# B&R Automation Studio project br_server
Automation Studio 4.4.6.71 SP

## Configuration minimal

### Task classes (Cpu.sw)
```
Cyclic#4:
  TCP_Server <- TcpIpServer.prg
Cyclic#7:
  ControlLoo <- ControlLoop.prg
Libraries: AsBrStr, AsIOTime, AsTCP, runtime, TcpIp, Transport
```

### Hardware
```
X20CP1586 : X20CP1586 v1.4.2.0
  Connector IF2:
    ActivateDevice = 1
    Mode = Manual
    InternetAddress = 10.4.22.176
    SubnetMask = 255.255.255.0
  ConfigurationID = br_server_minimal
  SimulationIPAddress = 10.4.22.176
```

## Logical view

Binary libraries used (declarations not repeated): operator, runtime, astime, AsIecCon, AsBrStr, AsIOTime, AsTCP

### Global.typ - Global data types
```iecst
TYPE
	_expData : 	STRUCT
		bActivateExperiment : BOOL;
	END_STRUCT;
	_trajData : 	STRUCT
		dStartValue : LREAL;
		lStartTime : UDINT;
		dEndValue : LREAL;
		lEndTime : UDINT;
		dOutput : LREAL;
	END_STRUCT;
	_benchData : 	STRUCT
		lTime : UDINT;
		dValue1 : LREAL;
		fValue2 : REAL;
		iValue3 : INT;
		cValue4 : BYTE;
	END_STRUCT;
	TcpServer_interface : 	STRUCT
		out_Encoder_Achse_1 : REAL;
		out_Encoder_Motor : REAL;
		out_Statusword : UINT;
		out_ActualValue : REAL;
		in_Controlword : UINT;
		in_Setpoint : REAL;
		tmp : ARRAY[0..3]OF USINT;
	END_STRUCT;
	TcpServer_instances : 	STRUCT
		TcpOpen_0 : TcpOpen;
		TcpServer_0 : TcpServer;
		TcpIoctl_0 : TcpIoctl;
		TcpRecv_0 : TcpRecv;
		TcpSend_0 : TcpSend;
		TcpClose_0 : TcpClose;
		linger_opt : tcpLINGER_typ;
	END_STRUCT;
END_TYPE
```

### Package Logical/Libraries - Global libraries

### Library Logical/Libraries/TcpIp (ANSIC)

#### TcpIpServer.cpp
```cpp
/** @file TcpIpServer.cpp
 *  @brief Implementation of the TcpIpServer Class
 */
#include "TcpIpServer.h"

#define LINGER_ON (1)

/**
*	@brief disable all function blocks
*/
void TcpIpServer::deinit()
{
	TcpClose_0.enable = false;
	TcpClose(&TcpClose_0);
	TcpOpen_0.enable = false;
	TcpOpen(&TcpOpen_0);
	TcpServer_0.enable = false;
	TcpServer(&TcpServer_0);
	TcpIoctl_0.enable = false;
	TcpIoctl(&TcpIoctl_0);
	TcpRecv_0.enable = false;
	TcpRecv(&TcpRecv_0);
	TcpSend_0.enable = false;
	TcpSend(&TcpSend_0);
	tcp_step = 0;
}

/**
*	@brief initialize server
*/
void TcpIpServer::init()
{
	this->_status = BUSY;
	static const struct tcpLINGER_typ linger_opt = {LINGER_ON, 0};
	switch(tcp_step) {
		case 0:
			deinit();
			tcp_step = 1;
			break;
		case 1:
			/* Open TCP Socket */
			TcpOpen_0.pIfAddr = 0;
			TcpOpen_0.port = this->serverPort;
			TcpOpen_0.options = tcpOPT_REUSEADDR;
			TcpOpen_0.enable = true;
			TcpOpen(&TcpOpen_0);
			if (TcpOpen_0.status == ERR_OK) {
				this->serverID = TcpOpen_0.ident;
				tcp_step = 2;
			} else if (TcpOpen_0.status == ERR_FUB_BUSY) {
				// intentionally blank
			} else {
				tcp_step = 0;
				this->_status = ERROR;
			}
			break;
		case 2:
			/* set server options */
			/* these ensure that the connection gets closed directly, without waiting for timeouts */
			/* see BuR AsTCP Help files for more information */

			TcpIoctl_0.ident = this->serverID;
			TcpIoctl_0.ioctl = tcpSO_LINGER_SET;
			TcpIoctl_0.pData = (unsigned long) &linger_opt;
			TcpIoctl_0.datalen = sizeof(linger_opt);
			TcpIoctl_0.enable = true;
			TcpIoctl(&TcpIoctl_0);
			if (TcpIoctl_0.status == ERR_OK) {
				//this->outlen = TcpIoctl_0.outlen;
				tcp_step = 3;
			} else if (TcpIoctl_0.status == ERR_FUB_BUSY) {
				// intentionally blank
			} else {
				tcp_step = 0;
				this->_status = ERROR;
			}
			break;
		case 3:
			/* start server and wait for client */
			TcpServer_0.ident = this->serverID;
			TcpServer_0.backlog = 1;
			TcpServer_0.pIpAddr = (unsigned long) this->clientIp;
			TcpServer_0.enable = true;
			TcpServer(&TcpServer_0);
			if (TcpServer_0.status == ERR_OK) {
				this->clientID = TcpServer_0.identclnt;
				//this->clientPort = TcpServer_0.portclnt;
				tcp_step = 4;
			} else if (TcpServer_0.status == ERR_FUB_BUSY) {
				//intentionally blank
			} else {
				tcp_step = 0;
				this->_status = ERROR;
			}
			break;
		case 4:
			/* set same options for client */
			TcpIoctl_0.ident = this->clientID;
			TcpIoctl_0.ioctl = tcpSO_LINGER_SET;
			TcpIoctl_0.pData = (unsigned long) &linger_opt;
			TcpIoctl_0.datalen = sizeof(linger_opt);
			TcpIoctl_0.enable = true;
			TcpIoctl(&TcpIoctl_0);
			if (TcpIoctl_0.status == ERR_OK) {
			//	this->client_outlen = TcpIoctl_0.outlen;
				this->_status = READY;
				tcp_step = 0;
			} else if (TcpIoctl_0.status == ERR_FUB_BUSY) {
				// intentionally blank
			} else {
				tcp_step = 0;
				this->_status = ERROR;
			}
			break;
		default:
			break;
	}
}

/**
 * @brief reads incoming data from client
 * data gets saved to inBuffer, the data length is written to inBufferLen
 */
TcpIpServer::Status TcpIpServer::read()
{
	TcpRecv_0.ident = this->clientID;
	TcpRecv_0.pData = (unsigned long) this->inBuffer;
	TcpRecv_0.datamax = sizeof(this->inBuffer);
	TcpRecv_0.flags = 0;
	TcpRecv_0.enable = true;
	TcpRecv(&TcpRecv_0);
	if (TcpRecv_0.status == ERR_OK)
	{
		this->inBufferLen = TcpRecv_0.recvlen;
		if (this->inBufferLen == 0)
		{
			/* client already disconnected */
			return STOP;
		}
		else
			return READY;
	}
	else if (TcpRecv_0.status == ERR_FUB_BUSY)
		;
	else if (TcpRecv_0.status == tcpERR_NO_DATA)
	{
		/* no data received */
		this->inBufferLen = 0;
		return READY;
	}
	else if (TcpRecv_0.status == tcpERR_NOT_CONNECTED)
	{
		/* connection closed */
		return STOP;
	}
	else
	{
		return ERROR;
	}
	return BUSY;
}

/**
 * @brief write data from the current outBuffer to the client
 */
TcpIpServer::Status TcpIpServer::write()
{
	TcpSend_0.ident = this->clientID;
	TcpSend_0.pData = (unsigned long) this->outBuffer;
	TcpSend_0.datalen = this->outBufferLen;
	TcpSend_0.flags = 0;
	TcpSend_0.enable = true;
	TcpSend(&TcpSend_0);
	if (TcpSend_0.status == ERR_OK)
	{
		this->outBufferLen = 0;
		return READY;
	}
	else if (TcpSend_0.status == ERR_FUB_BUSY)
		;
	else if (TcpSend_0.status == tcpERR_NOT_CONNECTED)
	{
		/* connection closed */
		return STOP;
	}
	else
		return ERROR;
	return BUSY;
}

void TcpIpServer::handleFrame(Frame frame)
{
	this->buffer_out[this->outc++] = frame.data.id;
	for (int i = 0; i < MAX_PAYLOAD; ++i) {
		this->buffer_out[this->outc++] = frame.data.payload[i];
	}
}

void TcpIpServer::sync()
{
	this->_status = BUSY;
	switch (tcp_step) {
		case 0:
			/**< Lese von Client*/
			this->_status_sub = read();
			switch (this->_status_sub) {
				case READY:
					if (this->inBufferLen > 0) {
						unsigned char *pointer = this->inBuffer;
						while (pointer - this->inBuffer < (signed long)this->inBufferLen) {
							Frame frame(pointer++[0]);
							for (int i = 0; i < MAX_PAYLOAD; ++i)
								frame.data.payload[i] = *pointer++;
							this->transp->handleFrame(frame);
						}
						this->inBufferLen = 0;
					}
					/**< Sende Daten falls vorhanden*/
					if (this->outBufferLen > 0) {
						tcp_step = 1;
					} else {
						tcp_step = 0;
						_status = READY;
					}
					break;
				case BUSY:
					// intentionally blank
					break;
				case STOP:
					tcp_step = 0;
					_status = STOP;
					break;
				default:
					tcp_step = 0;
					_status = ERROR;
					break;
			}
			break;
		case 1:
			/**< Schreibe Daten an Client*/
			_status_sub = write();
			switch (_status_sub) {
				case READY:
					tcp_step = 0;
					_status = READY;
					break;
				case BUSY:
					// intentionally blank
					break;
				case STOP:
					tcp_step = 0;
					_status = STOP;
					break;
				default:
					tcp_step = 0;
					_status = ERROR;
					break;
			}
			break;
		default:
			break;
	}
}

void TcpIpServer::closeSockets()
{
	_status = BUSY;
	switch (tcp_step)
	{
		case 0:
			/**< Schließe Client Socket*/
			TcpClose_0.ident = this->clientID;
			TcpClose_0.how = 0;
			TcpClose_0.enable = true;
			TcpClose(&TcpClose_0);
			if (TcpClose_0.status == ERR_OK)
			{
				tcp_step = 1;
			}
			else if (TcpClose_0.status == ERR_FUB_BUSY)
				;
			else
			{
				tcp_step = 255;
				_status = ERROR;
			}
			break;
		case 1:
			/**< Schließe Server*/
			TcpClose_0.ident = this->serverID;
			TcpClose_0.how = 0;
			TcpClose_0.enable = true;
			TcpClose(&TcpClose_0);
			if (TcpClose_0.status == ERR_OK)
			{
				_status = READY;
				tcp_step = 0;
			}
			else if (TcpClose_0.status == ERR_FUB_BUSY)
				;
			else
			{
				tcp_step = 255;
				_status = ERROR;
			}
			break;
		default:
			break;
	}
}

void TcpIpServer::registerListener(Comm *t)
{
	this->transp = t;
}

void TcpIpServer::resetBuffs(void)
{
	this->outBufferLen = 0;
	this->inBufferLen = 0;
	for (int i = 0; i < 255 * (MAX_PAYLOAD + 1); ++i) {
		this->outBuffer[i] = 0;
		this->inBuffer[i] = 0;
	}
}
```

#### TcpIpServer.h
```c
#ifndef TCPSERVER_CLASS_H
#define TCPSERVER_CLASS_H
#include <bur/plctypes.h>
#ifdef _DEFAULT_INCLUDES
#include <AsDefault.h>
#endif
#include <AsTCP.h>
#include <AsIOTime.h>
#include "../Comm.h"
#include "../Transport/Frame.h"

/** @file TcpServer.h
 *  @class TcpIpServer
 *  @brief Implementation of a simple TCP Server
 *
 *	The server is initialised and run using the AsTCP library.
 */

class TcpIpServer: public Comm{
	public:
	/** server status enum */
	enum Status
	{
		ERROR = 0xFF,
		STOP = 0,
		BUSY,
		READY
	};
	private:
	const int serverPort;		///< port to be used by the server
	unsigned long serverID;		///< server ID for function blocks
	//unsigned long outlen;
	unsigned long clientIp;		///< IP address of connected client
	unsigned long clientID;		///< client ID for function blocks
	//unsigned int clientPort;	///< port of client
	//unsigned long client_outlen;

	unsigned short tcp_step;		///< step variable for the server state-machine

	Status _status;
	Status _status_sub;

	struct TcpOpen TcpOpen_0;
	struct TcpServer TcpServer_0;
	struct TcpIoctl TcpIoctl_0;
	struct TcpRecv TcpRecv_0;
	struct TcpSend TcpSend_0;
	struct TcpClose TcpClose_0;

	unsigned char outBuffer[255 * (MAX_PAYLOAD + 1)];
	unsigned int outBufferLen;
	unsigned char inBuffer[255 * (MAX_PAYLOAD + 1)];
	unsigned int inBufferLen;
	/**< Tcp read und write Funktionen*/
	Status read();
	Status write();

	Comm *transp;

	public:
	TcpIpServer(int port)
		:serverPort(port),
		status(_status)
	{};
	/**< Initialisierungsmethode*/
	void deinit();
	void init();
	/**< Zyklische Lese- und Schreibmethode*/
	void sync();
	/**< Schließen der Sockets*/
	void closeSockets();
	/**< Readonly methode um Status zu lesen*/
	const Status &status;
	/** Method to queue communication frame */
	void handleFrame(Frame frame);
	/** Method to register the transport protocol instance */
	void registerListener(Comm *transp);
	/** Method to reset buffers upon experiment end */
	void resetBuffs(void);
};
#endif //TCPSERVER_CLASS_H
```

### Library Logical/Libraries/Transport (ANSIC)

#### Transport.h
```c
#ifndef TRANSPORT_CLASS_H
#define TRANSPORT_CLASS_H

#include "../Comm.h"
#include "Frame.h"
/** \file Transport.h
 *  \class Transport
 *  \brief Klasse zum Ent- und Packen der Kommunikationsdaten zu Pywisp
 *
 *  Die Klasse wird mit zwei Buffer initialisiert, einen Eingangsbuffer und
 *  einen Ausgangsbuffer. Diese Buffer müssen die gleiche Länge besitzen wie
 *  die auf Pywisp. Will man mehrere Frames schicken, so können weitere Buffer
 *  über die addOutBuffer() Methode hinzugefügt werden. Damit diese auch
 *  gesendet werden, muss entsprechender Frame in sendData() gepackt werden.
 *  Eingangsseitig gibt es nur einen Buffer der die Frames liefert. Mit
 *  der Methode run() kann kontrolliert werden, ob Eingangsseitig Daten
 *  ausgewertet werden müssen. Mittels runExp() kann kontrolliert werden
 *  ob ein Experiment ausgeführt werden soll.
 */

class Transport: public Comm {
	public:
	void handleFrame(Frame frame);

	void sendData();

	void registerServer(Comm *serv);

	private:
	Comm *tcp;

	void unpackExp(Frame frame);

	void unpackBenchData(Frame frame);

	void unpackTrajRampData(Frame frame);

};

extern Transport transport;

#endif //TRANSPORT_CLASS_H
```

#### Transport.cpp
```cpp
#define _BUR_USE_DECLARATION_IN_IEC
#ifdef _DEFAULT_INCLUDES
#include "AsDefault.h"
#endif
#include "Transport.h"

/**
 * @brief Method that defines and sends all testbench frames
 */
void Transport::sendData() {
	Frame benchFrame(10);
	benchFrame.pack(benchData.lTime);
	benchFrame.pack(benchData.dValue1);
	benchFrame.pack(benchData.fValue2);
	benchFrame.pack(benchData.iValue3);
	benchFrame.pack(benchData.cValue4);
	tcp->handleFrame(benchFrame);

	Frame trajFrame(11);
	trajFrame.pack(benchData.lTime);
	trajFrame.pack(trajData.dOutput);
	tcp->handleFrame(trajFrame);
}

/*
 * @brief handles all frames arriving at the testbench
 */
void Transport::handleFrame(Frame frame)
{
	switch (frame.data.id) {
		case 1:
			unpackExp(frame);
			break;
		case 12:
			unpackBenchData(frame);
			break;
		case 13:
			unpackTrajRampData(frame);
			break;
		default:;
	}
}

/**
 * @brief unpacks experiment activation status and resets experiment time
 */
void Transport::unpackExp(Frame frame) {
	frame.unPack(expData.bActivateExperiment);
	benchData.lTime = 0;
}

void Transport::unpackBenchData(Frame frame) {
	frame.unPack(benchData.dValue1);
	frame.unPack(benchData.fValue2);
	frame.unPack(benchData.iValue3);
	frame.unPack(benchData.cValue4);
}

void Transport::unpackTrajRampData(Frame frame) {
	frame.unPack(trajData.dStartValue);
	frame.unPack(trajData.lStartTime);
	frame.unPack(trajData.dEndValue);
	frame.unPack(trajData.lEndTime);
}

/**
 * @brief registers Server for handling outgoing frames
 */
void Transport::registerServer(Comm *serv)
{
	this->tcp = serv;
}
```

#### Frame.h
```c
/** @file Frame.h
 *
 */
#ifndef FRAME_H
#define FRAME_H

#include <bur/plctypes.h>
#ifdef _DEFAULT_INCLUDES
#include <AsDefault.h>
#endif
#include <stdint.h>

#include "../Comm.h"

/**
 * Class, that implements a byte wise frame that is interchanged by connection. The frame has an id and a payload
 * for the specific data. The data is stored as an byte array. It implements all functions to store and unpack
 * the data to and from byte wise array. The id represents the identification of the frame.
 */
class Frame {

public:
	struct _data {
		unsigned char id;
		unsigned char payload[80];
	} data;

	Frame(unsigned char id) {
		data.id = id;
		cCursor = 0;
	}

	Frame() {
		cCursor = 0;
	}

    /**
     * Adds a double value to payload
     * @param dValue value that is packed in payload
     */
	void pack(double dValue) {
		uPack.dVar = dValue;
		for (int i = 0; i < 8; ++i)
			data.payload[cCursor + i] = uPack.cVar[7 - i];

		cCursor += 8;
	};

    /**
     * Adds an unsigned long value to payload
     * @param lValue value that is packed in payload
     */
	void pack(unsigned long lValue) {
		data.payload[cCursor + 0] = (unsigned char) ((lValue & 0xff000000UL) >> 24);
		data.payload[cCursor + 1] = (unsigned char) ((lValue & 0x00ff0000UL) >> 16);
		data.payload[cCursor + 2] = (unsigned char) ((lValue & 0x0000ff00UL) >> 8);
		data.payload[cCursor + 3] = (unsigned char) (lValue & 0x000000ffUL);

		cCursor += 4;
	};

    /**
     * Adds a float value to payload
     * @param fValue value that is packed in payload
     */
	void pack(float fValue) {
		uPack.fVar1 = fValue;
		for (int i = 0; i < 4; ++i)
			data.payload[cCursor + i] = uPack.cVar[7 - i];

		cCursor += 4;
	};

    /**
     * Adds an integer value to payload
     * @param iValue value that is packed in payload
     */
	void pack(int iValue) {
		data.payload[cCursor + 0] = (unsigned char) ((iValue & 0x0000ff00UL) >> 8);
		data.payload[cCursor + 1] = (unsigned char) (iValue & 0x000000ffUL);

		cCursor += 2;
	};

    /**
     * Adds an unsigned char value to payload
     * @param cValue value that is packed in payload
     */
	void pack(unsigned char cValue) {
		data.payload[cCursor + 0] = cValue;

		cCursor++;
	};

    /**
     * Return a double value from payload
     * @param dValue value with unpacked data
     */
	void unPack(double &dValue) {
		for (int i = 0; i < 8; ++i)
			uPack.cVar[7 - i] = data.payload[cCursor + i];
		dValue = uPack.dVar;

		cCursor += 8;
	};

    /**
     * Return an unsigned long value from payload
     * @param lValue value with unpacked data
     */
	void unPack(unsigned long &lValue) {
		lValue = ((uint32_t) (data.payload[cCursor + 0]) << 24) |
			((uint32_t) (data.payload[cCursor + 1]) << 16) |
			((uint32_t) (data.payload[cCursor + 2]) << 8) |
			(uint32_t) (data.payload[cCursor + 3]);

		cCursor += 4;
	};

    /**
     * Return a float value from payload
     * @param fValue value with unpacked data
     */
	void unPack(float &fValue) {
		for (int i = 0; i < 4; ++i)
			uPack.cVar[7 - i] = data.payload[cCursor + i];
		fValue = uPack.fVar1;

		cCursor += 4;
	};

    /**
     * Return an integer value from payload
     * @param iValue value with unpacked data
     */
	void unPack(int &iValue) {
		iValue = ((uint32_t) (data.payload[cCursor + 0]) << 8) |
			(uint32_t) (data.payload[cCursor + 1]);

		cCursor += 2;
	};

	/**
     * Return an integer value from payload
     * @param iValue value with unpacked data
     */
	void unPack(short &iValue) {
		iValue = ((uint32_t) (data.payload[cCursor + 0]) << 8) |
			(uint32_t) (data.payload[cCursor + 1]);

		cCursor += 2;
	};

    /**
     * Return an unsigned char value from payload
     * @param cValue value with unpacked data
     */
	void unPack(unsigned char &cValue) {
		cValue = data.payload[cCursor + 0];

		cCursor++;
	};

    /**
     * Return a bool value from payload
     * @param bValue value with unpacked data
     */
	void unPack(bool &bValue) {
		bValue = data.payload[cCursor + 0];

		cCursor++;
	};

private:
	unsigned char cCursor;

	union {
		double dVar;
		struct {
			float fVar2;
			float fVar1;
		};
		unsigned char cVar[8];
	} uPack;

};

#endif //SERVER_FRAME_H
```

### Comm.h
```c
#ifndef COMM_H
#define COMM_H

#include "Frame/Frame.h"

#define MAX_PAYLOAD (80)

class Comm {
public:
	virtual void handleFrame(Frame frame) = 0;
};

#endif
```

### Library Logical/Libraries/Frame (ANSIC)

#### Frame.h
```c
/** @file Frame.h
 *
 */
#ifndef FRAME_H
#define FRAME_H

#include <bur/plctypes.h>
#ifdef _DEFAULT_INCLUDES
#include <AsDefault.h>
#endif
#include <stdint.h>

#include "../Comm.h"

/**
 * Class, that implements a byte wise frame that is interchanged by connection. The frame has an id and a payload
 * for the specific data. The data is stored as an byte array. It implements all functions to store and unpack
 * the data to and from byte wise array. The id represents the identification of the frame.
 */
class Frame {

public:
	struct _data {
		unsigned char id;
		unsigned char payload[80];
	} data;

	Frame(unsigned char id) {
		data.id = id;
		cCursor = 0;
	}

	Frame() {
		cCursor = 0;
	}

    /**
     * Adds a double value to payload
     * @param dValue value that is packed in payload
     */
	void pack(double dValue) {
		uPack.dVar = dValue;
		for (int i = 0; i < 8; ++i)
			data.payload[cCursor + i] = uPack.cVar[7 - i];

		cCursor += 8;
	};

    /**
     * Adds an unsigned long value to payload
     * @param lValue value that is packed in payload
     */
	void pack(unsigned long lValue) {
		data.payload[cCursor + 0] = (unsigned char) ((lValue & 0xff000000UL) >> 24);
		data.payload[cCursor + 1] = (unsigned char) ((lValue & 0x00ff0000UL) >> 16);
		data.payload[cCursor + 2] = (unsigned char) ((lValue & 0x0000ff00UL) >> 8);
		data.payload[cCursor + 3] = (unsigned char) (lValue & 0x000000ffUL);

		cCursor += 4;
	};

    /**
     * Adds a float value to payload
     * @param fValue value that is packed in payload
     */
	void pack(float fValue) {
		uPack.fVar1 = fValue;
		for (int i = 0; i < 4; ++i)
			data.payload[cCursor + i] = uPack.cVar[7 - i];

		cCursor += 4;
	};

    /**
     * Adds an integer value to payload
     * @param iValue value that is packed in payload
     */
	void pack(int iValue) {
		data.payload[cCursor + 0] = (unsigned char) ((iValue & 0x0000ff00UL) >> 8);
		data.payload[cCursor + 1] = (unsigned char) (iValue & 0x000000ffUL);

		cCursor += 2;
	};

    /**
     * Adds an unsigned char value to payload
     * @param cValue value that is packed in payload
     */
	void pack(unsigned char cValue) {
		data.payload[cCursor + 0] = cValue;

		cCursor++;
	};

    /**
     * Return a double value from payload
     * @param dValue value with unpacked data
     */
	void unPack(double &dValue) {
		for (int i = 0; i < 8; ++i)
			uPack.cVar[7 - i] = data.payload[cCursor + i];
		dValue = uPack.dVar;

		cCursor += 8;
	};

    /**
     * Return an unsigned long value from payload
     * @param lValue value with unpacked data
     */
	void unPack(unsigned long &lValue) {
		lValue = ((uint32_t) (data.payload[cCursor + 0]) << 24) |
			((uint32_t) (data.payload[cCursor + 1]) << 16) |
			((uint32_t) (data.payload[cCursor + 2]) << 8) |
			(uint32_t) (data.payload[cCursor + 3]);

		cCursor += 4;
	};

    /**
     * Return a float value from payload
     * @param fValue value with unpacked data
     */
	void unPack(float &fValue) {
		for (int i = 0; i < 4; ++i)
			uPack.cVar[7 - i] = data.payload[cCursor + i];
		fValue = uPack.fVar1;

		cCursor += 4;
	};

    /**
     * Return an integer value from payload
     * @param iValue value with unpacked data
     */
	void unPack(int &iValue) {
		iValue = ((uint32_t) (data.payload[cCursor + 0]) << 8) |
			(uint32_t) (data.payload[cCursor + 1]);

		cCursor += 2;
	};

    /**
     * Return an unsigned char value from payload
     * @param cValue value with unpacked data
     */
	void unPack(unsigned char &cValue) {
		cValue = data.payload[cCursor + 0];

		cCursor++;
	};

    /**
     * Return a bool value from payload
     * @param bValue value with unpacked data
     */
	void unPack(bool &bValue) {
		bValue = data.payload[cCursor + 0];

		cCursor++;
	};

private:
	unsigned char cCursor;

	union {
		double dVar;
		struct {
			float fVar2;
			float fVar1;
		};
		unsigned char cVar[8];
	} uPack;

};

#endif //SERVER_FRAME_H
```

### Library Logical/Libraries/TCPServer (ANSIC)

#### TCPServer.cpp
```cpp
#include "TCPServer.h"

/** \file TCPServer.cpp
 *  \brief Implementation der TCPServer Klasse
 */
void TCPServer::deinit()
{
	/**< Clearen aller Funktionsblöcke*/
	TcpClose_0.enable = false;
	TcpClose(&TcpClose_0);
	TcpOpen_0.enable = false;
	TcpOpen(&TcpOpen_0);
	TcpServer_0.enable = false;
	TcpServer(&TcpServer_0);
	TcpIoctl_0.enable = false;
	TcpIoctl(&TcpIoctl_0);
	TcpRecv_0.enable = false;
	TcpRecv(&TcpRecv_0);
	TcpSend_0.enable = false;
	TcpSend(&TcpSend_0);
	tcp_step = 0;
}

void TCPServer::init()
{
	this->_status = BUSY;
	switch(tcp_step) {
		case 0:
			deinit();
			tcp_step = 1;
			break;
		case 1:
			/**< Öffnen des Tcp Sockets*/
			TcpOpen_0.pIfAddr = 0; //(unsigned long) this->server_ip;
			TcpOpen_0.port = this->server_port;
			TcpOpen_0.options = tcpOPT_REUSEADDR;
			TcpOpen_0.enable = true;
			TcpOpen(&TcpOpen_0);
			if (TcpOpen_0.status == ERR_OK) {
				this->ident = TcpOpen_0.ident;
				//TcpOpen_0->enable = false;
				tcp_step = 2;
			} else if (TcpOpen_0.status == ERR_FUB_BUSY) {
				// intentionally blank
			} else {
				tcp_step = 0;
				this->_status = ERROR;
			}
			break;
		case 2:
			/**< Nimm Einstellungen vor, siehe Hilfe von AsTCP*/
			/**< Durch diese Einstellung wird die Verbindung direkt abgebrochen ohne Buffer zu leeren*/
			linger_opt.lLinger = 0;
			linger_opt.lOnOff = 1;

			TcpIoctl_0.ident = this->ident;
			TcpIoctl_0.ioctl = tcpSO_LINGER_SET;
			TcpIoctl_0.pData = (unsigned long) &this->linger_opt;
			TcpIoctl_0.datalen = this->linger_opt_len;
			TcpIoctl_0.enable = true;
			TcpIoctl(&TcpIoctl_0);
			if (TcpIoctl_0.status == ERR_OK) {
				this->outlen = TcpIoctl_0.outlen;
				//TcpIoctl_0->enable = false;
				tcp_step = 3;
			} else if (TcpIoctl_0.status == ERR_FUB_BUSY) {
				// intentionally blank
			} else {
				tcp_step = 0;
				this->_status = ERROR;
			}
			break;
		case 3:
			/**< Starte den Server und warte auf Client*/
			TcpServer_0.ident = ident;
			TcpServer_0.backlog = 1;
			TcpServer_0.pIpAddr = (unsigned long) this->client_ip;
			TcpServer_0.enable = true;
			TcpServer(&TcpServer_0);
			if (TcpServer_0.status == ERR_OK) {
				this->client_ident = TcpServer_0.identclnt;
				this->client_port = TcpServer_0.portclnt;
				//TcpServer_0->enable = false;
				tcp_step = 4;
			} else if (TcpServer_0.status == ERR_FUB_BUSY) {
				//intentionally blank
			} else {
				tcp_step = 0;
				this->_status = ERROR;
			}
			break;
		case 4:
			/**< Gleiche Einstellungen für Client*/
			TcpIoctl_0.ident = this->client_ident;
			TcpIoctl_0.ioctl = tcpSO_LINGER_SET;
			TcpIoctl_0.pData = (unsigned long) &this->linger_opt;
			TcpIoctl_0.datalen = this->linger_opt_len;
			TcpIoctl_0.enable = true;
			TcpIoctl(&TcpIoctl_0);
			if (TcpIoctl_0.status == ERR_OK) {
				this->client_outlen = TcpIoctl_0.outlen;
				//TcpIoctl_0->enable = false;
				this->_status = READY;
				tcp_step = 0;
			} else if (TcpIoctl_0.status == ERR_FUB_BUSY) {
				// intentionally blank
			} else {
				tcp_step = 0;
				this->_status = ERROR;
			}
			break;
		default:
			break;
	}
}

TCPServer::Status TCPServer::read()
{
	/**< Lese von Client*/
	TcpRecv_0.ident = this->client_ident;
	TcpRecv_0.pData = (unsigned long) this->buffer_in;
	TcpRecv_0.datamax = sizeof(this->buffer_in);
	TcpRecv_0.flags = 0;
	TcpRecv_0.enable = true;
	TcpRecv(&TcpRecv_0);
	if (TcpRecv_0.status == ERR_OK)
	{
		this->recvlength = TcpRecv_0.recvlen;
		//TcpRecv_0->enable = false;
		if (this->recvlength == 0)
		{
			/**< Client bereits geschlossen*/
			return STOP;
		}
		else
			return READY;
	}
	else if (TcpRecv_0.status == ERR_FUB_BUSY)
		;
	else if (TcpRecv_0.status == tcpERR_NO_DATA)
	{
		/**< Keine Daten empfangen*/
		this->recvlength = 0;
		//TcpRecv_0->enable = false;
		return READY;
	}
	else if (TcpRecv_0.status == tcpERR_NOT_CONNECTED)
	{
		/**< Verbindung wurde getrennt*/
		//TcpRecv_0->enable = false;
		return STOP;
	}
	else
	{
		return ERROR;
	}
	return BUSY;
}

TCPServer::Status TCPServer::write()
{
	/**< Schreibe Daten an Client*/
	TcpSend_0.ident = client_ident;
	TcpSend_0.pData = (unsigned long) buffer_out;
	TcpSend_0.datalen = (MAX_PAYLOAD + 1) * outc;
	TcpSend_0.flags = 0;
	TcpSend_0.enable = true;
	TcpSend(&TcpSend_0);
	outc = 0;
	if (TcpSend_0.status == ERR_OK)
	{
		//TcpSend_0->enable = false;
		return READY;
	}
	else if (TcpSend_0.status == ERR_FUB_BUSY)
		;
	else if (TcpSend_0.status == tcpERR_NOT_CONNECTED)
	{
		/**< Verbindung wurde getrennt*/
		//TcpSend_0->enable = false;
		return STOP;
	}
	else
		return ERROR;
	return BUSY;
}

void TCPServer::handleFrame(Frame frame)
{
	this->buffer_out[this->outc].data.id = frame.data.id;
	for (int i = 0; i < MAX_PAYLOAD; ++i) {
		this->buffer_out[this->outc].data.payload[i] =frame.data.payload[i];
	}
	this->outc++;
}

void TCPServer::sync()
{
	this->_status = BUSY;
	switch (tcp_step) {
		case 0:
			/**< Lese von Client*/
			this->_status_sub = read();
			switch (this->_status_sub) {
				case READY:
					if (this->recvlength > 0) {
						unsigned char *pointer = buffer_in;
						while (pointer - buffer_in < this->recvlength) {
							Frame frame(pointer++[0]);
							for (int i = 0; i < MAX_PAYLOAD; ++i)
								frame.data.payload[i] = *pointer++;
							this->transp->handleFrame(frame);
						}
						recvlength = 0;
					}
					/**< Sende Daten falls vorhanden*/
					if (this->outc > 0) {
						tcp_step = 1;
					} else {
						tcp_step = 0;
						_status = READY;
					}
					break;
				case BUSY:
					// intentionally blank
					break;
				case STOP:
					tcp_step = 0;
					_status = STOP;
					break;
				default:
					tcp_step = 0;
					_status = ERROR;
					break;
			}
			break;
		case 1:
			/**< Schreibe Daten an Client*/
			_status_sub = write();
			switch (_status_sub) {
				case READY:
					tcp_step = 0;
					_status = READY;
					break;
				case BUSY:
					// intentionally blank
					break;
				case STOP:
					tcp_step = 0;
					_status = STOP;
					break;
				default:
					tcp_step = 0;
					_status = ERROR;
					break;
			}
			break;
		default:
			break;
	}
}

void TCPServer::close_sockets()
{
	_status = BUSY;
	switch (tcp_step)
	{
		case 0:
			/**< Schließe Client Socket*/
			TcpClose_0.ident = client_ident;
			TcpClose_0.how = 0;
			TcpClose_0.enable = true;
			TcpClose(&TcpClose_0);
			if (TcpClose_0.status == ERR_OK)
			{
				//TcpClose_0->enable = false;
				tcp_step = 1;
			}
			else if (TcpClose_0.status == ERR_FUB_BUSY)
				;
			else
			{
				tcp_step = 255;
				_status = ERROR;
			}
			break;
		case 1:
			/**< Schließe Server*/
			TcpClose_0.ident = ident;
			TcpClose_0.how = 0;
			TcpClose_0.enable = true;
			TcpClose(&TcpClose_0);
			if (TcpClose_0.status == ERR_OK)
			{
				// TcpClose_0->enable = false;
				_status = READY;
				tcp_step = 0;
			}
			else if (TcpClose_0.status == ERR_FUB_BUSY)
				;
			else
			{
				tcp_step = 255;
				_status = ERROR;
			}
			break;
		default:
			break;
	}
}

void TCPServer::registerListener(Comm *t)
{
	transp = t;
}
```

#### TCPServer.h
```c
#ifndef TCPSERVER_CLASS_H
#define TCPSERVER_CLASS_H
#include <bur/plctypes.h>
#ifdef _DEFAULT_INCLUDES
#include <AsDefault.h>
#endif
#include <AsTCP.h>
#include <AsIOTime.h>
#include "../Comm.h"
#include "../Frame/Frame.h"

/** \file TCPServer.h
 *  \class TCPServer
 *  \brief Klasse Aufsetzen eines TCP Servers
 *
 *  Über die AsTCP Bibliothek wird der TCP Server initialisiert und ausgeführt.
 *  Die Funktionsblöcke werden als Pointer der Klasse übergeben und im Code
 *  aufgerufen. Zudem wird der Eventlogger verwendet, um evtl. Fehler zu loggen.
 */

class TCPServer: public Comm{
	public:
	/** Status definition der Klasse*/
	enum Status
	{
		ERROR = 0xFF,
		STOP = 0,
		BUSY,
		READY
	};
	private:
	/* Variablen für Verbindungsparameter*/
	const int server_port;
	unsigned long ident;
	unsigned long outlen;
	unsigned long client_ip;
	unsigned long client_ident;
	unsigned int client_port;
	unsigned long client_outlen;

	unsigned short tcp_step;
	/* Statusvariablen*/
	Status _status;
	Status _status_sub;
	/* Pointer auf Funktionsblöcke*/
	struct TcpOpen TcpOpen_0;
	struct TcpServer TcpServer_0;
	struct TcpIoctl TcpIoctl_0;
	struct TcpRecv TcpRecv_0;
	struct TcpSend TcpSend_0;
	struct TcpClose TcpClose_0;
	struct tcpLINGER_typ linger_opt;
	unsigned int linger_opt_len;
	/**< Sende- und Empfangsbuffer mit Längen und cursor*/
	Frame buffer_out[255];
	unsigned int outc;
	unsigned char buffer_in[255 * (MAX_PAYLOAD + 1)];
	unsigned int recvlength;
	/**< Tcp read und write Funktionen*/
	Status read();
	Status write();

	Comm *transp;

	public:
	TCPServer(int port)
		:server_port(port),
		status(_status)
	{};
	/**< Initialisierungsmethode*/
	void deinit();
	void init();
	/**< Zyklische Lese- und Schreibmethode*/
	void sync();
	/**< Schließen der Sockets*/
	void close_sockets();
	/**< Readonly methode um Status zu lesen*/
	const Status &status;
	/** Method to queue communication frame */
	void handleFrame(Frame frame);
	void registerListener(Comm *transp);
};
#endif //TCPSERVER_CLASS_H
```

### Program Logical/TCP_Server (ANSIC)

#### Main.cpp
```cpp
#define _BUR_USE_DECLARATION_IN_IEC
#ifdef _DEFAULT_INCLUDES
	#include "AsDefault.h"
#endif
#include "../Libraries/TCPServer/TCPServer.h"
#include "../Libraries/Transport/Transport.h"

/**< amount of memory to be allocated for heap storage must be specified for
     every ANSI C++ program with the bur_heap_size variable */
unsigned long bur_heap_size = 0xFFFFF;

/**< Zählervariablen*/
int counter_close = 0;
int counter_tcp = 0;
/**< Instanz der Tcp Server Klasse*/
TCPServer TCPS_0(50007);

/**< Instanz der Transport Klasse*/
Transport transport;

void _INIT ProgramInit(void)
{
	Main_state = 0;
	counter_close = 0;
	counter_tcp = 0;
	TCPS_0.registerListener(&transport);
	transport.registerServer(&TCPS_0);
	TCPS_0.deinit();
	for (long int i = 0; i < 0xFFFFFFFF; ++i)
		;

}

void _CYCLIC ProgramCyclic(void)
{
    switch (Main_state)
    {
        case 0:
            /**< Starte Server und warte auf Client*/
            TCPS_0.init();
            if (TCPS_0.status == TCPServer::READY)
				;//Main_state = 1; TODO DEBUG
            else if ((TCPS_0.status == TCPServer::STOP) || (TCPS_0.status == TCPServer::ERROR))
				;//Main_state = 255; TODO DEBUG
            break;
        case 1:
            /**< Lese und Schreibe mit Client*/
            TCPS_0.sync();
            if (TCPS_0.status == TCPServer::READY)
				Main_state = 1;
            else if ((TCPS_0.status == TCPServer::STOP) || (TCPS_0.status == TCPServer::ERROR))
				Main_state = 10;
            break;
        case 10:
            /**< Schließe Verbindung*/
            TCPS_0.close_sockets();
            if (TCPS_0.status == TCPServer::READY)
                Main_state = 11;
            break;
        case 11:
            /**< Warte 5 Sekunden und starte Server erneut*/
            if (counter_close > 500)
            {
                counter_close = 0;
                Main_state = 0;
            }
            else
                counter_close += 1;
            break;
        default:
            break;
    }
	if (expData.bActivateExperiment) {
		if (counter_tcp >= 10) {
			transport.sendData();
			counter_tcp = 0;
		} else {
			counter_tcp += 1;
		}
	}
}

void _EXIT ProgramExit(void)
{
	// Insert code here
    TCPS_0.close_sockets();
}
```

### Program Logical/ControlLoop (ANSIC)

#### Main.cpp
```cpp
#include <bur/plc.h>
#include <bur/plctypes.h>
#ifdef _DEFAULT_INCLUDES
	#include <AsDefault.h>
#endif

#include "../Libraries/Transport/Transport.h"

// amount of memory to be allocated for heap storage must be specified for every ANSI C++ program with the bur_heap_size variable
unsigned long bur_heap_size = 0xFFFF;
const unsigned long lDt = 1000;          ///< Sampling step [ms]

/**
 * @brief Method that calculates a trajectory value and writes the return value in _trajData->dOutput
 * @param _benchData pointer to test rig data struct
 * @param _trajData pointer to trajectory struct
 */
void fTrajectory() {
	if ( benchData.lTime < trajData.lStartTime ) {
		trajData.dOutput = trajData.dStartValue;
	} else {
		if (benchData.lTime < trajData.lEndTime) {
			double dM = (trajData.dEndValue - trajData.dStartValue) / (trajData.lEndTime - trajData.lStartTime);
			double dN = trajData.dEndValue - dM * trajData.lEndTime;
			trajData.dOutput = dM * benchData.lTime + dN;
		} else {
			trajData.dOutput = trajData.dEndValue;
		}
	}
}

void _INIT ProgramInit(void)
{
	benchData.lTime = 0;
	benchData.dValue1 = 0;
	benchData.fValue2 = 0;
	benchData.iValue3 = 0;
	benchData.cValue4 = 0;

	trajData.dStartValue = 0;
	trajData.lStartTime = 0;
	trajData.dEndValue = 0;
	trajData.lEndTime = 0;
	trajData.dOutput = 0;
}

void _CYCLIC ProgramCyclic(void)
{
	if (expData.bActivateExperiment) {
		benchData.lTime += lDt;

		fTrajectory();
	}
}

void _EXIT ProgramExit(void)
{
	// Insert code here

}
```

### Program Logical/TcpIpServer

#### Variables.var
```iecst
VAR
	mainState : USINT := 0;
END_VAR
```

#### Main.cpp
```cpp
#define _BUR_USE_DECLARATION_IN_IEC
#ifdef _DEFAULT_INCLUDES
	#include "AsDefault.h"
#endif
#include "../Libraries/TcpIp/TcpIpServer.h"
#include "../Libraries/Transport/Transport.h"

/**< amount of memory to be allocated for heap storage must be specified for
     every ANSI C++ program with the bur_heap_size variable */
unsigned long bur_heap_size = 0xFFFFF;

/**< Zählervariablen*/
int counter_close = 0;
int counter_tcp = 0;
/**< Instanz der Tcp Server Klasse*/
TcpIpServer TCPS_0(50007);

/**< Instanz der Transport Klasse*/
Transport transport;

void _INIT ProgramInit(void)
{
	Main_state = 0;
	counter_close = 0;
	counter_tcp = 0;
	TCPS_0.registerListener(&transport);
	transport.registerServer(&TCPS_0);
	TCPS_0.deinit();
}

void _CYCLIC ProgramCyclic(void)
{
	switch (Main_state)
	{
		case 0:
			/**< Starte Server und warte auf Client*/
			TCPS_0.init();
			if (TCPS_0.status == TcpIpServer::READY)
				Main_state = 1;
			else if ((TCPS_0.status == TcpIpServer::STOP) || (TCPS_0.status == TcpIpServer::ERROR))
				Main_state = 255;
			break;
		case 1:
			/**< Lese und Schreibe mit Client*/
			TCPS_0.sync();
			if (TCPS_0.status == TcpIpServer::READY)
				Main_state = 1;
			else if ((TCPS_0.status == TcpIpServer::STOP) || (TCPS_0.status == TcpIpServer::ERROR))
				Main_state = 10;
			break;
		case 10:
			/**< Schließe Verbindung*/
			TCPS_0.close_sockets();
			if (TCPS_0.status == TcpIpServer::READY)
				Main_state = 11;
			break;
		case 11:
			/**< Warte 5 Sekunden und starte Server erneut*/
			if (counter_close > 50)
			{
				counter_close = 0;
				Main_state = 0;
			}
			else
				counter_close += 1;
			break;
		default:
			break;
	}
	/**< Sende alle 100 ms Messdaten zu Pywisp*/
	if (expData.bActivateExperiment) {
		transport.sendData();
		benchData.lTime += 100;
	}
}

void _EXIT ProgramExit(void)
{
    TCPS_0.close_sockets();
}
```

Listed in the project but not available here: Logical/Global.var
